// TwinCAT 3 PLC project PLC
// ProgramVersion: 3.1.4024.0
// libraries:
//   Tc2_MC2, * (Beckhoff Automation GmbH)
//   Tc2_Standard, * (Beckhoff Automation GmbH)
//   Tc2_System, * (Beckhoff Automation GmbH)
//   Tc3_Module, * (Beckhoff Automation GmbH)
// project tree:
//   DUTs/ data.TcDUT
//   GVLs/ GVL.TcGVL
//   / PlcTask.TcTTO
//   POUs/ fbAbsolute.TcPOU, MAIN.TcPOU

CONFIGURATION PLC
    RESOURCE PLC ON TwinCAT3
        TASK PlcTask(INTERVAL := T#10ms, PRIORITY := 20);
        PROGRAM MAIN WITH PlcTask : MAIN;
    END_RESOURCE
END_CONFIGURATION

// ---- DUTs/data.TcDUT
TYPE data :
STRUCT
	boEnable 		:BOOL;
	boStart 		:BOOL;
	lrPosition  	:LREAL;
	lrVelocity  	:LREAL;
	lrAcceleration 	:LREAL;
	lrDeceleration 	:LREAL;
	lrJerk 			:LREAL;
	
	lrActualPos 	:LREAL;
	lrActualVelo	:LREAL;
	lrActualAcc 	:LREAL;
END_STRUCT
END_TYPE

// ---- GVLs/GVL.TcGVL
{attribute 'qualified_only'}
VAR_GLOBAL
	stData	:data;
END_VAR

// ---- POUs/MAIN.TcPOU
PROGRAM MAIN
VAR
	fbMotor: fbAbsolute;
	
	fbPower		:mc_Power;
	fbAbsolute  :mc_MoveAbsolute;
	axis		:axis_ref;
	
	ftrboEnable	:f_trig;
END_VAR


gvl.stData.lrActualPos:=axis.NcToPlc.ActPos;
gvl.stData.lrActualVelo:=axis.NcToPlc.ActVelo;
gvl.stData.lrActualAcc:=axis.NcToPlc.ActAcc;

fbMotor(
	boEnable:=gvl.stData.boEnable , 
	boStart:=gvl.stData.boStart , 
	lrPos:=gvl.stData.lrPosition , 
	lrVelo:=gvl.stData.lrVelocity , 
	lrAcc:=gvl.stData.lrAcceleration , 
	lrDec:=gvl.stData.lrDeceleration , 
	lrJerk:=gvl.stData.lrJerk , 
	fbPower:=fbPower , 
	fbAbsolute:=fbAbsolute , 
	axis:=axis );
	
IF fbAbsolute.Done THEN
	gvl.stData.boStart:=false;
END_IF 

ftrboEnable(CLK:=gvl.stData.boEnable);

IF ftrboEnable.Q THEN
	gvl.stData.boStart:=false;
END_IF

END_PROGRAM

// ---- POUs/fbAbsolute.TcPOU
FUNCTION_BLOCK fbAbsolute
VAR_INPUT
	boEnable	:BOOL;
	boStart		:BOOL;
	
	lrPos		:LREAL;
	lrVelo		:LREAL;
	lrAcc		:LREAL;
	lrDec		:LREAL;
	lrJerk		:LREAL;
END_VAR
VAR_OUTPUT
END_VAR
VAR
	iState		:INT:=0;
	sState		:STRING;
	rtrboStart	:R_trig;
	ftrboEnable	:f_trig;
	tonMoveNotDone	:ton;
END_VAR
VAR_IN_OUT
	fbPower		:mc_Power;
	fbAbsolute  :mc_MoveAbsolute;
	axis		:axis_ref;
END_VAR


rtrboStart(CLK:=boStart);
ftrboEnable(CLK:=boEnable);

CASE iState OF
0:
	IF boEnable THEN
		iState:=100;
	END_IF
100:
	IF rtrboStart.Q THEN
		fbAbsolute.Execute:=TRUE;
		tonMoveNotDone.IN:=TRUE;
		iState:=1000;
	END_IF
1000:
	fbAbsolute.Execute:=FALSE;
	IF fbAbsolute.Done  THEN
		tonMoveNotDone.IN:=FALSE;
		iState:=100;
	ELSIF tonMoveNotDone.Q THEN
		sState:='motor dont have achived target position';
		tonMoveNotDone.IN:=FALSE;
		iState:=100;
	END_IF	
END_CASE

tonMoveNotDone(PT:=T#100s);

IF ftrboEnable.Q THEN
	iState:=0;
	sState:='';
	fbAbsolute.Execute:=FALSE;
	tonMoveNotDone.IN:=FALSE;
END_IF

fbPower(
	Axis:=axis , 
	Enable:=boEnable , 
	Enable_Positive:=boEnable , 
	Enable_Negative:=boEnable , 
	Override:=100);
	
fbAbsolute(
	Axis:=axis , 
	Position:=lrPos , 
	Velocity:=lrVelo , 
	Acceleration:=lrAcc , 
	Deceleration:=lrDec , 
	Jerk:=lrJerk  );

END_FUNCTION_BLOCK
